FUNCTION_BLOCK Lift (* Composite Function Block Type *)
  (* Standard: 61499-2 *)
  (* Version 0.0, 6/3/2016, Andrei, nxtControl GmbH, template *)
  PACKAGE Main;
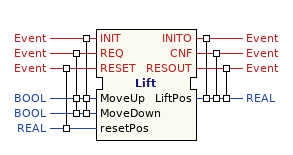
  EVENT_INPUT
    INIT WITH MoveUp, MoveDown; (* Initialization Request *)
    REQ WITH MoveUp, MoveDown; (* Normal Execution Request *)
    RESET WITH resetPos;
  END_EVENT
  EVENT_OUTPUT
    INITO WITH LiftPos; (* Initialization Confirm *)
    CNF WITH LiftPos; (* Execution Confirmation *)
    RESOUT WITH LiftPos;
  END_EVENT
  VAR_INPUT
    MoveUp : BOOL; (* Input event qualifier *)
    MoveDown : BOOL;
    resetPos : REAL;
  END_VAR
  VAR_OUTPUT
    LiftPos : REAL; (* Output event qualifier *)
  END_VAR
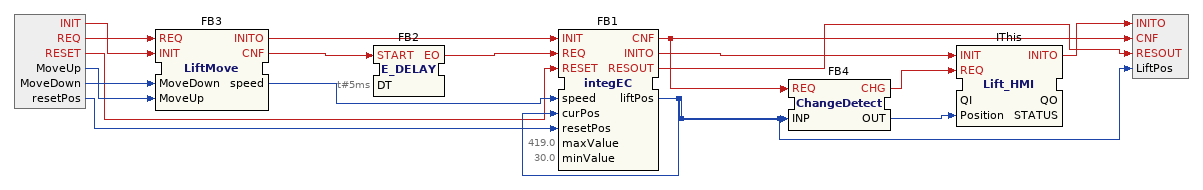
  FBS
    FB4 : ChangeDetect;
    IThis : Lift_HMI;
    FB2 : E_DELAY(DT := t#5ms);
    FB3 : LiftMove;
    FB1 : integEC(maxValue := 419.0, minValue := 30.0);
  END_FBS
  EVENT_CONNECTIONS
    REQ TO FB3.REQ;
    INIT TO FB3.INIT;
    FB3.INITO TO FB1.INIT;
    FB1.CNF TO FB4.REQ;
    FB1.CNF TO CNF;
    FB2.EO TO FB1.REQ;
    FB3.CNF TO FB2.START;
    FB1.INITO TO IThis.INIT;
    FB4.CHG TO IThis.REQ;
    IThis.INITO TO INITO;
    RESET TO FB1.RESET;
    FB1.RESOUT TO RESOUT;
  END_CONNECTIONS
  DATA_CONNECTIONS
    FB3.speed TO FB1.speed;
    MoveDown TO FB3.MoveDown;
    MoveUp TO FB3.MoveUp;
    FB1.liftPos TO FB4.INP;
    FB1.liftPos TO LiftPos;
    FB1.liftPos TO FB1.curPos;
    FB4.OUT TO IThis.Position;
    resetPos TO FB1.resetPos;
  END_CONNECTIONS
END_FUNCTION_BLOCK
